PROGRAM MAIN
VAR
stThisIsOurFirstInstanceOfAStructure : ST_Event;
bBoolean : BOOL := FALSE;
fFahrenheit : REAL ;
nReturnGreater: INT ;
nReturnSmaller : INT;

nA : INT := 5 ;
nB : INT := 15;

END_VAR


fFahrenheit := Celcius_to_Fahrenet(fCelcius:= 5.0) ;

Greater_Smaller (nNumber1:=8,
	             nNumber2:=15,
				 nGreater => nReturnGreater,
				 nSmaller=>nReturnSmaller );			 
SwapNums(nNumber3 := nA, 
		 nNumber4 := nB);
		 
IF NOT bBoolean THEN
UpdateEventTimeStampWithSystemTime(ST_Event := stThisIsOurFirstInstanceOfAStructure);
bBoolean:= TRUE;
	
END_IF

END_PROGRAM

(* stored: Version 1.1.0.1, ProductVersion 3.1.4024.9
   POU MAIN: Id {bdc4ab82-e035-4559-afb2-1b6836e8376d}, SpecialFunc None *)
